{attribute 'qualified_only'}
VAR_GLOBAL
	Ax		:axis_ref;
END_VAR

(* stored: Version 1.1.0.1, ProductVersion 3.1.4024.12
   GVL GVL: Id {cc519fc8-fa47-4117-8109-d071c0f4a902} *)
